(* IEC 61131-3 sources: BODAS-HelloWorld/extracted_st/bodas_rc18_12_40/plc_logic/application/01_maintask/02_outputs/prg_safeouts, 1 file *)

(* ---- PRG_SafeOuts.st ---- *)
(* --- Interface --- *)
(*********************************************************************************************************************
*    __   __   ___  ___           __   __        __   __  ___
*   /_ / /  / /__  /    /__/     /_ / /_   |_ / /_ / /  /  /  /__/
*  /__/ /__/ __ / /__  /  /     /  | /__  /  | /  | /__/  /  /  /
*
* Project: Hello World for ml290.rts
*
* Program: PRG_Outputs
*
* Author:
*
* Description:
* Interface for the hardware outputs to the application
*
* (c) Copyright by BOSCH REXROTH AG, all rights reserved
*
*********************************************************************************************************************)
PROGRAM PRG_SafeOuts
VAR
    PHMDL_CHNL1 : UINT := UDINT_TO_UINT(PHMDL OR CHNL1);
END_VAR
